// TIA Portal V17 export
// export: Created 2022-07-20T06:59:49.6889473Z, ExportSetting WithDefaults, DisplayName Totally Integrated Automation Portal, DisplayVersion V17, DisplayName TIA Portal Openness, DisplayVersion V17, DisplayName TIA Portal Version Control Interface, DisplayVersion V17, DisplayName SINAMICS Startdrive Advanced, DisplayVersion V17, DisplayName SINAMICS Startdrive G130, G150, S120, S150, SINAMICS MV, S210, DisplayVersion V17, DisplayName SINAMICS Startdrive G110M, G120, G120C, G120D, G120P, G115D, DisplayVersion V17, DisplayName STEP 7 Professional, DisplayVersion V17, DisplayName STEP 7 Safety, DisplayVersion V17, DisplayName WinCC Advanced, DisplayVersion V17
FUNCTION "FC10023_ParameterBoundariesCheck" : Void   // FC10023, LAD
{ S7_Optimized_Access := 'TRUE' }
VERSION : 0.1
// stored: AutoNumber false, IsIECCheckEnabled false, SetENOAutomatically false, UDAEnableTagReadback false
   VAR_INPUT
      LowerBoundary : LReal;
      UpperBoundary : LReal;
      Parameter : LReal;
   END_VAR
   VAR_OUTPUT
      LowerBoundaryExceeded : Bool;
      LowerBoundaryNotAllowed : Bool;
      UpperBoundaryExceeded : Bool;
      UpperBoundaryNotAllowed : Bool;
   END_VAR
BEGIN

REGION Network 1 (SCL): Boundaries Check
   IF
       (#UpperBoundary < #LowerBoundary) OR
       (#UpperBoundary = #LowerBoundary AND #LowerBoundary = 0.0)
   THEN
       #LowerBoundaryNotAllowed := TRUE;
       #UpperBoundaryNotAllowed := TRUE;
   ELSE
       #LowerBoundaryNotAllowed := FALSE;
       #UpperBoundaryNotAllowed := FALSE;
   END_IF;
END_REGION

REGION Network 2 (SCL): Paramerters Boundaries Management
   IF #Parameter < #LowerBoundary THEN
       #LowerBoundaryExceeded := TRUE;
   ELSE
       #LowerBoundaryExceeded := FALSE;
   END_IF;

   IF #Parameter > #UpperBoundary THEN
       #UpperBoundaryExceeded := TRUE;
   ELSE
       #UpperBoundaryExceeded := FALSE;
   END_IF;
END_REGION
END_FUNCTION
